// TIA Portal project "Process Control 1" (V13)

(* hardware
DEVICE "S71500/ET200MP station_1"  S7-1500 station
   slot 0: "导轨_0"  6ES7 590-1***0-0AA0
   slot 1: "PLC_1"  CPU 1516-3 PN/DP  6ES7 516-3AN00-0AB0  V1.8
   slot 2: "DI 32x24VDC HF_1"  DI 32x24VDC HF  6ES7 521-1BL00-0AB0  V2.0
   slot 3: "DQ 32x24VDC/0.5A ST_1"  DQ 32x24VDC/0.5A ST  6ES7 522-1BL00-0AB0  V2.0
   slot 4: "AI 8xU/I/RTD/TC ST_1"  AI 8xU/I/RTD/TC ST  6ES7 531-7KF00-0AB0  V2.0
   slot 5: "AQ 4xU/I ST_1"  AQ 4xU/I ST  6ES7 532-5HD00-0AB0  V2.0
DEVICE "PC-System_1"  SIMATIC PC station
   slot 0: "SIMATIC PC station"  Rail  SIMATIC PC-Station  V1.0
      slot 125: "Stationmanager"  Station_Manager  V6.0.4
   slot 1: "HMI_RT_1"  WinCC RT Advanced  6AV2 104-0xxxx-xxxx  13.0.1.0
      slot 33792: "主机接口"  主机接口
   slot 2: "IE general_1"  IE General  IE_CP  V8.2.0
*)

// ===== PLC "PLC_1"  CPU 1516-3 PN/DP =====

VAR_GLOBAL   // PLC tag table "默认变量表"
   "Tag_1" AT %IW4 : Word;
   "Tag_2" AT %MD0 : Real;
   "Tag_3" AT %MD4 : Real;
   "Tag_4" AT %MD8 : Real;
   "Tag_5" AT %MD12 : Real;
   "Tag_6" AT %QW4 : Int;
   "exp_sel01" AT %M16.0 : Bool;
   "exp_sel02" AT %M16.1 : Bool;
   "Tag_7" AT %IW6 : Int;
END_VAR

DATA_BLOCK "TO_WINCC_01"   // DB2
{ S7_Optimized_Access := 'FALSE' }
VERSION : 0.1
   VAR
      Level_Setpoint : Real;
      Level_Feedback : Real;
      Valve_Output : Real;
      Input_sel : Bool;
      ManualValue : Real;
      PID_Reset : Bool;
      PID_Mode : Int;
      Gain : Real;
      Ti : Real;
      Td : Real;
      exp_sel01 : Bool;
      exp_sel02 : Bool;
      Auto_state : Bool;
      Manual_state : Bool;
      Manual_Auto : Bool;
   END_VAR
BEGIN
END_DATA_BLOCK

DATA_BLOCK "TO_WINCC_02"   // DB3
{ S7_Optimized_Access := 'FALSE' }
VERSION : 0.1
   VAR
      Gain_内环 : Real;
      Ti_内环 : Real;
      Gain_外环 : Real;
      Ti_外环 : Real;
      Td_外环 : Real;
   END_VAR
BEGIN
END_DATA_BLOCK

FUNCTION "过控实验1" : Void   // FC1, LAD
{ S7_Optimized_Access := 'FALSE' }
VERSION : 0.1
BEGIN

REGION Network 1: activate peripheral input
   // 选择INPUT或者INPUT_PER参数，为0时是INPUT，为1时是INPUT_PER
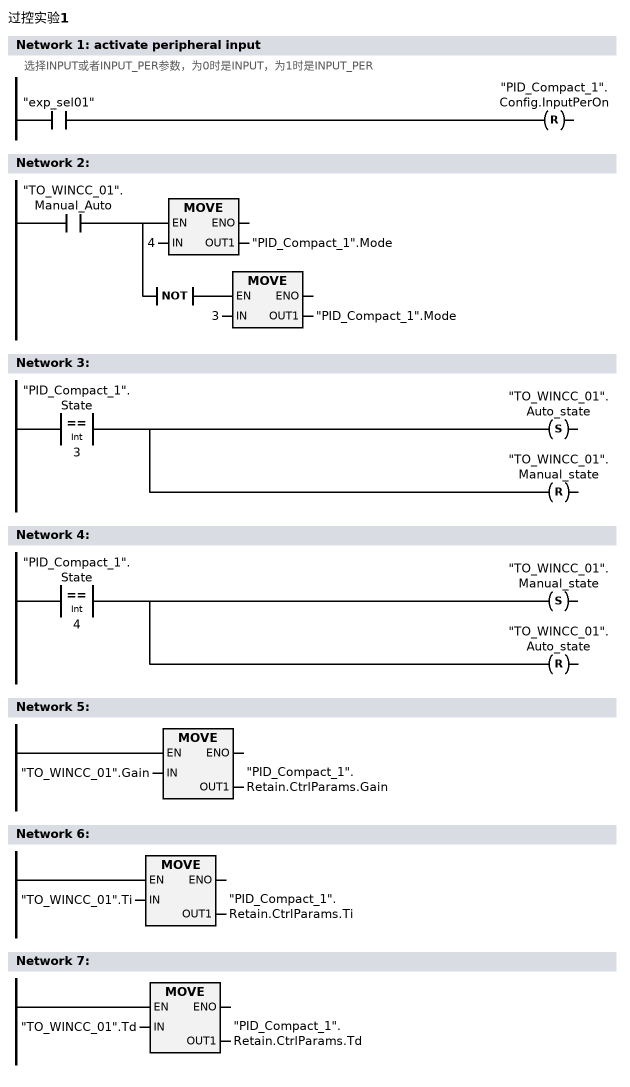
   RUNG wire#powerrail
      Contact( "exp_sel01" )
      R_Coil( "PID_Compact_1".Config.InputPerOn )
   END_RUNG
   // the same network as SCL:
   IF "exp_sel01" THEN "PID_Compact_1".Config.InputPerOn := FALSE; END_IF;
END_REGION

REGION Network 2
   RUNG wire#powerrail
      Contact( "TO_WINCC_01".Manual_Auto )
      wire#w1
      Move(in := 4, out1 => "PID_Compact_1".Mode)
   END_RUNG
   RUNG wire#w1
      Not()
      Move(in := 3, out1 => "PID_Compact_1".Mode)
   END_RUNG
   // the same network as SCL:
   IF "TO_WINCC_01".Manual_Auto THEN "PID_Compact_1".Mode := 4; END_IF;
   IF NOT "TO_WINCC_01".Manual_Auto THEN "PID_Compact_1".Mode := 3; END_IF;
END_REGION

REGION Network 3
   RUNG wire#powerrail
      { S7_Templates := "SrcType := Int" } EQ_Contact(in1 := "PID_Compact_1".State, in2 := 3)
      wire#w1
      S_Coil( "TO_WINCC_01".Auto_state )
   END_RUNG
   RUNG wire#w1
      R_Coil( "TO_WINCC_01".Manual_state )
   END_RUNG
   // the same network as SCL:
   IF "PID_Compact_1".State = 3 THEN
       "TO_WINCC_01".Auto_state := TRUE;
       "TO_WINCC_01".Manual_state := FALSE;
   END_IF;
END_REGION

REGION Network 4
   RUNG wire#powerrail
      { S7_Templates := "SrcType := Int" } EQ_Contact(in1 := "PID_Compact_1".State, in2 := 4)
      wire#w1
      S_Coil( "TO_WINCC_01".Manual_state )
   END_RUNG
   RUNG wire#w1
      R_Coil( "TO_WINCC_01".Auto_state )
   END_RUNG
   // the same network as SCL:
   IF "PID_Compact_1".State = 4 THEN
       "TO_WINCC_01".Manual_state := TRUE;
       "TO_WINCC_01".Auto_state := FALSE;
   END_IF;
END_REGION

REGION Network 5
   RUNG wire#powerrail
      Move(in := "TO_WINCC_01".Gain, out1 => "PID_Compact_1".Retain.CtrlParams.Gain)
   END_RUNG
   // the same network as SCL:
   "PID_Compact_1".Retain.CtrlParams.Gain := "TO_WINCC_01".Gain;
END_REGION

REGION Network 6
   RUNG wire#powerrail
      Move(in := "TO_WINCC_01".Ti, out1 => "PID_Compact_1".Retain.CtrlParams.Ti)
   END_RUNG
   // the same network as SCL:
   "PID_Compact_1".Retain.CtrlParams.Ti := "TO_WINCC_01".Ti;
END_REGION

REGION Network 7
   RUNG wire#powerrail
      Move(in := "TO_WINCC_01".Td, out1 => "PID_Compact_1".Retain.CtrlParams.Td)
   END_RUNG
   // the same network as SCL:
   "PID_Compact_1".Retain.CtrlParams.Td := "TO_WINCC_01".Td;
END_REGION
END_FUNCTION

FUNCTION "过控实验2" : Void   // FC2, LAD
{ S7_Optimized_Access := 'FALSE' }
VERSION : 0.1
BEGIN

REGION Network 1: activate peripheral input
   // 选择INPUT或者INPUT_PER参数，为0时是INPUT，为1时是INPUT_PER
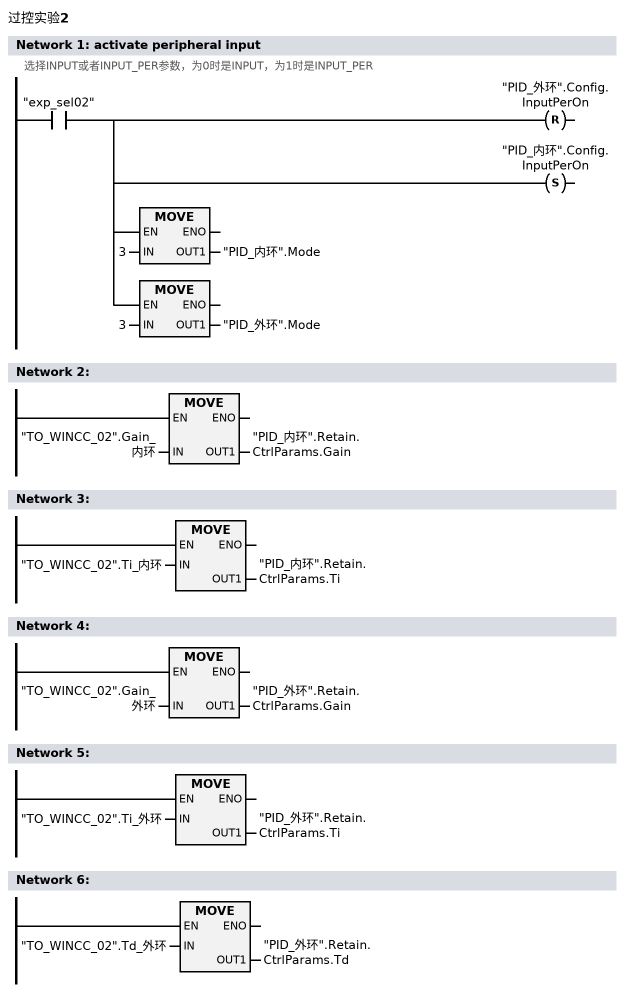
   RUNG wire#powerrail
      Contact( "exp_sel02" )
      wire#w1
      R_Coil( "PID_外环".Config.InputPerOn )
   END_RUNG
   RUNG wire#w1
      S_Coil( "PID_内环".Config.InputPerOn )
   END_RUNG
   RUNG wire#w1
      Move(in := 3, out1 => "PID_内环".Mode)
   END_RUNG
   RUNG wire#w1
      Move(in := 3, out1 => "PID_外环".Mode)
   END_RUNG
   // the same network as SCL:
   IF "exp_sel02" THEN
       "PID_外环".Config.InputPerOn := FALSE;
       "PID_内环".Config.InputPerOn := TRUE;
       "PID_内环".Mode := 3;
       "PID_外环".Mode := 3;
   END_IF;
END_REGION

REGION Network 2
   RUNG wire#powerrail
      Move(in := "TO_WINCC_02".Gain_内环, out1 => "PID_内环".Retain.CtrlParams.Gain)
   END_RUNG
   // the same network as SCL:
   "PID_内环".Retain.CtrlParams.Gain := "TO_WINCC_02".Gain_内环;
END_REGION

REGION Network 3
   RUNG wire#powerrail
      Move(in := "TO_WINCC_02".Ti_内环, out1 => "PID_内环".Retain.CtrlParams.Ti)
   END_RUNG
   // the same network as SCL:
   "PID_内环".Retain.CtrlParams.Ti := "TO_WINCC_02".Ti_内环;
END_REGION

REGION Network 4
   RUNG wire#powerrail
      Move(in := "TO_WINCC_02".Gain_外环, out1 => "PID_外环".Retain.CtrlParams.Gain)
   END_RUNG
   // the same network as SCL:
   "PID_外环".Retain.CtrlParams.Gain := "TO_WINCC_02".Gain_外环;
END_REGION

REGION Network 5
   RUNG wire#powerrail
      Move(in := "TO_WINCC_02".Ti_外环, out1 => "PID_外环".Retain.CtrlParams.Ti)
   END_RUNG
   // the same network as SCL:
   "PID_外环".Retain.CtrlParams.Ti := "TO_WINCC_02".Ti_外环;
END_REGION

REGION Network 6
   RUNG wire#powerrail
      Move(in := "TO_WINCC_02".Td_外环, out1 => "PID_外环".Retain.CtrlParams.Td)
   END_RUNG
   // the same network as SCL:
   "PID_外环".Retain.CtrlParams.Td := "TO_WINCC_02".Td_外环;
END_REGION
END_FUNCTION

FUNCTION "块_1" : Void   // FC3, LAD
{ S7_Optimized_Access := 'FALSE' }
VERSION : 0.1
BEGIN
END_FUNCTION

ORGANIZATION_BLOCK "Main"   // OB1, LAD, ProgramCycle
TITLE = "Main Program Sweep (Cycle)"
{ S7_Optimized_Access := 'FALSE' }
VERSION : 0.1
BEGIN
END_ORGANIZATION_BLOCK

ORGANIZATION_BLOCK "Cyclic interrupt"   // OB30, LAD, CyclicInterrupt
{ S7_Optimized_Access := 'FALSE' }
VERSION : 0.1
   VAR_TEMP   // added for the SCL form of the ladder/FBD networks
      _w1 : Bool;
   END_VAR
BEGIN

REGION Network 1
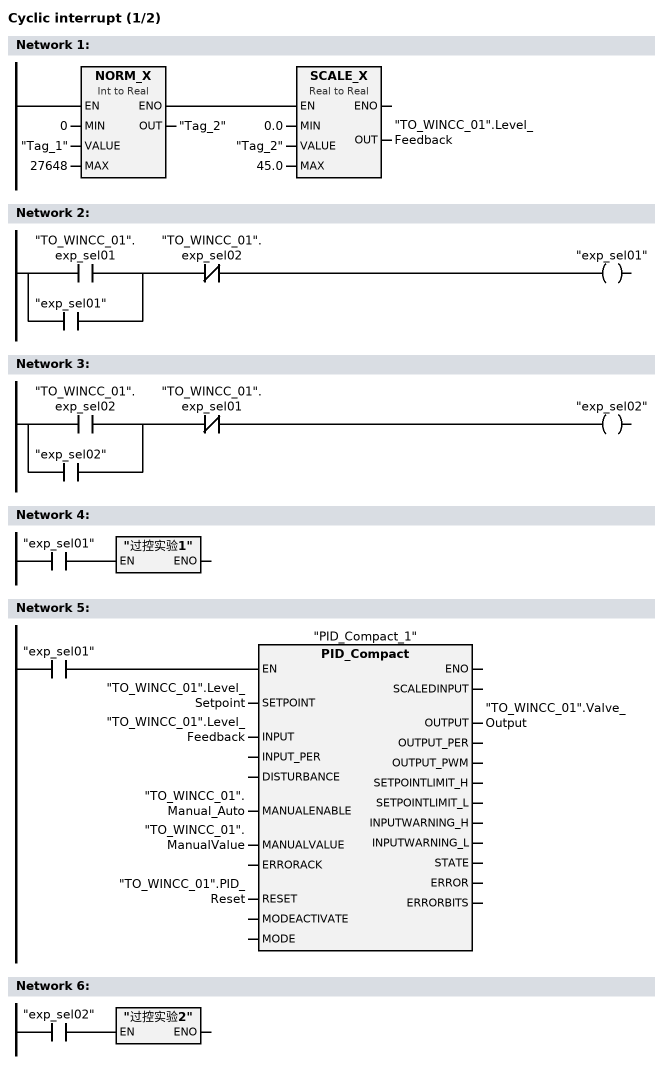
   RUNG wire#powerrail
      { S7_Templates := "[SrcType := Int, DestType := Real]" } Normalize(min := 0, value := "Tag_1", max := 27648, out => "Tag_2")
      { S7_Templates := "[SrcType := Real, DestType := Real]" } Scale(min := 0.0, value := "Tag_2", max := 45.0, out => "TO_WINCC_01".Level_Feedback)
   END_RUNG
   // the same network as SCL:
   "Tag_2" := NORM_X(MIN := 0, VALUE := "Tag_1", MAX := 27648);
   "TO_WINCC_01".Level_Feedback := SCALE_X(MIN := 0.0, VALUE := "Tag_2", MAX := 45.0);
END_REGION

REGION Network 2
   RUNG wire#powerrail
      Contact( "TO_WINCC_01".exp_sel01 )
      wire#w1
      I_Contact( "TO_WINCC_01".exp_sel02 )
      Coil( "exp_sel01" )
   END_RUNG
   RUNG wire#powerrail
      Contact( "exp_sel01" )
   END_RUNG wire#w1
   // the same network as SCL:
   "exp_sel01" := ("TO_WINCC_01".exp_sel01 OR "exp_sel01") AND NOT "TO_WINCC_01".exp_sel02;
END_REGION

REGION Network 3
   RUNG wire#powerrail
      Contact( "TO_WINCC_01".exp_sel02 )
      wire#w1
      I_Contact( "TO_WINCC_01".exp_sel01 )
      Coil( "exp_sel02" )
   END_RUNG
   RUNG wire#powerrail
      Contact( "exp_sel02" )
   END_RUNG wire#w1
   // the same network as SCL:
   "exp_sel02" := ("TO_WINCC_01".exp_sel02 OR "exp_sel02") AND NOT "TO_WINCC_01".exp_sel01;
END_REGION

REGION Network 4
   RUNG wire#powerrail
      Contact( "exp_sel01" )
      "过控实验1"()
   END_RUNG
   // the same network as SCL:
   IF "exp_sel01" THEN "过控实验1"(); END_IF;
END_REGION

REGION Network 5
   IF "exp_sel01" THEN
       "PID_Compact_1"(Setpoint := "TO_WINCC_01".Level_Setpoint,   // PID_Compact
                       Input := "TO_WINCC_01".Level_Feedback,
                       ManualEnable := "TO_WINCC_01".Manual_Auto,
                       ManualValue := "TO_WINCC_01".ManualValue,
                       Reset := "TO_WINCC_01".PID_Reset,
                       Output => "TO_WINCC_01".Valve_Output);
   END_IF;
END_REGION

REGION Network 6
   RUNG wire#powerrail
      Contact( "exp_sel02" )
      "过控实验2"()
   END_RUNG
   // the same network as SCL:
   IF "exp_sel02" THEN "过控实验2"(); END_IF;
END_REGION

REGION Network 7
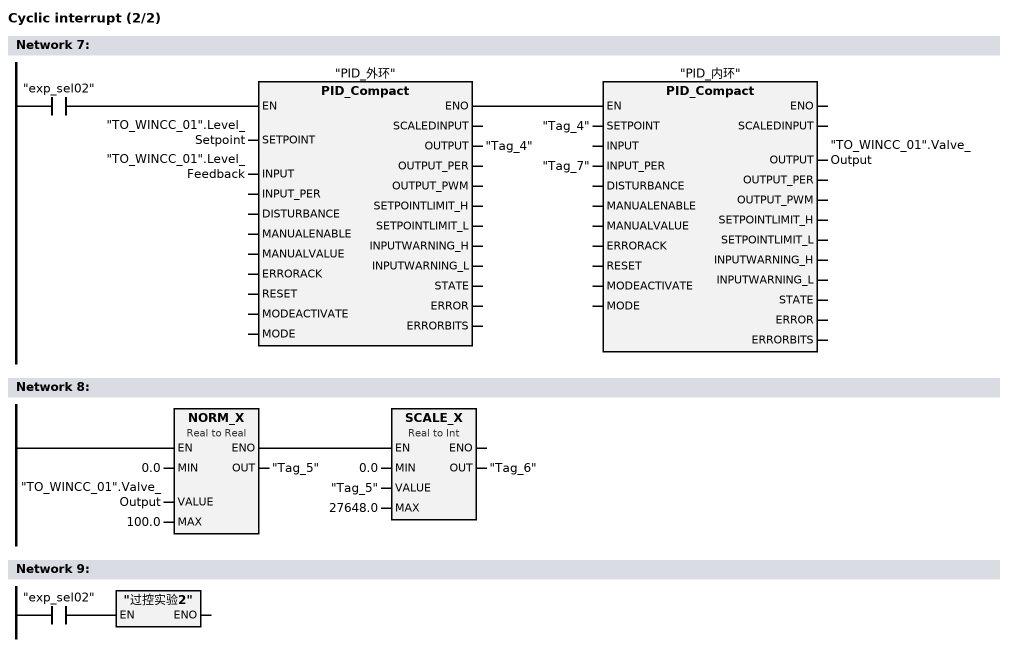
   // ENO of a box is taken as its EN; it also drops when the box reports an error
   #_w1 := "exp_sel02";
   IF #_w1 THEN
       "PID_外环"(Setpoint := "TO_WINCC_01".Level_Setpoint, Input := "TO_WINCC_01".Level_Feedback, Output => "Tag_4");   // PID_Compact
       "PID_内环"(Setpoint := "Tag_4", Input_PER := "Tag_7", Output => "TO_WINCC_01".Valve_Output);   // PID_Compact
   END_IF;
END_REGION

REGION Network 8
   RUNG wire#powerrail
      { S7_Templates := "[SrcType := Real, DestType := Real]" } Normalize(min := 0.0, value := "TO_WINCC_01".Valve_Output, max := 100.0, out => "Tag_5")
      { S7_Templates := "[SrcType := Real, DestType := Int]" } Scale(min := 0.0, value := "Tag_5", max := 27648.0, out => "Tag_6")
   END_RUNG
   // the same network as SCL:
   "Tag_5" := NORM_X(MIN := 0.0, VALUE := "TO_WINCC_01".Valve_Output, MAX := 100.0);
   "Tag_6" := SCALE_X(MIN := 0.0, VALUE := "Tag_5", MAX := 27648.0);
END_REGION

REGION Network 9
   RUNG wire#powerrail
      Contact( "exp_sel02" )
      "过控实验2"()
   END_RUNG
   // the same network as SCL:
   IF "exp_sel02" THEN "过控实验2"(); END_IF;
END_REGION
END_ORGANIZATION_BLOCK

(* ===== HMI "HMI_RT_1" =====
connection "HMI_连接_1": ETHERNET, S7_1500_OMS

HMI tags "默认变量表"
   "TO_WINCC_exp_sel01" : Bool, 100 ms
   "TO_WINCC_exp_sel02" : Bool, 100 ms
   "TO_WINCC_Level_Setpoint" : Real, 100 ms
   "TO_WINCC_Level_Feedback" : Real, 100 ms
   "TO_WINCC_Gain" : Real, 100 ms
   "TO_WINCC_Manual_Auto" : Bool, 100 ms
   "TO_WINCC_ManualValue" : Real, 100 ms
   "TO_WINCC_Manual_state" : Bool, 100 ms
   "TO_WINCC_Auto_state" : Bool, 100 ms
   "TO_WINCC_Ti" : Real, 100 ms
   "TO_WINCC_Td" : Real, 100 ms
   "TO_WINCC_Valve_Output" : Real, 100 ms
   "TO_WINCC_02_Gain_内环" : Real, 100 ms
   "TO_WINCC_02_Ti_内环" : Real, 100 ms
   "TO_WINCC_02_Gain_外环" : Real, 100 ms
   "TO_WINCC_02_Ti_外环" : Real, 100 ms
   "TO_WINCC_02_Td_外环" : Real, 100 ms
   "Tag_4" : Real = PLC "Tag_4", 100 ms
   "Tag_7" : Int = PLC "Tag_7", 100 ms
   "exp_sel01" : Bool = PLC "exp_sel01", 100 ms
   "exp_sel02" : Bool = PLC "exp_sel02", 100 ms

screen "实验选择主画面" 1600x1200
   TextField "文本域_1" at 326,82 size 878x101
   Button "按钮_1" at 498,276 size 562x118
   Button "按钮_2" at 498,501 size 562x118
   TextField "文本域_2" at 390,730 size 785x68

screen "实验1" 1600x1200
   TextField "文本域_1" at 595,12 size 338x40
   TextField "文本域_2" at 27,84 size 150x31
   IOField "I/O 域_1" at 187,80 size 165x36
   TextField "文本域_3" at 414,81 size 150x31
   IOField "I/O 域_2" at 590,79 size 165x36
   TextField "文本域_4" at 126,129 size 49x31
   IOField "I/O 域_3" at 187,126 size 165x36
   TextField "文本域_5" at 1196,30 size 20x31
   Button "按钮_1" at 1268,125 size 230x36
   TextField "文本域_6" at 1249,79 size 137x31
   TextField "文本域_7" at 1389,79 size 63x31
   TextField "文本域_8" at 1196,29 size 150x31
   IOField "I/O 域_4" at 1375,28 size 165x36
   TextField "文本域_9" at 1451,79 size 63x31
   TextField "文本域_10" at 1388,79 size 63x31
   TextField "文本域_11" at 442,129 size 123x31
   IOField "I/O 域_5" at 590,124 size 165x36
   TextField "文本域_12" at 924,128 size 49x31
   IOField "I/O 域_6" at 1002,124 size 165x36
   TrendView "趋势视图_1" at 15,195 size 1562x614
   TextField "文本域_13" at 824,80 size 150x31
   IOField "I/O 域_7" at 1001,78 size 165x36
   TextField "文本域_14" at 27,12 size 179x31
   TextField "文本域_15" at 27,12 size 179x31

screen "实验2" 1600x1200
   TextField "文本域_1" at 595,10 size 338x40
   TextField "文本域_14" at 206,83 size 150x31
   IOField "I/O 域_8" at 366,79 size 165x36
   TextField "文本域_15" at 593,82 size 150x31
   IOField "I/O 域_9" at 769,78 size 165x36
   TextField "文本域_2" at 1004,79 size 150x31
   IOField "I/O 域_1" at 1181,77 size 165x36
   TextField "文本域_3" at 247,137 size 107x31
   IOField "I/O 域_2" at 366,134 size 165x36
   TextField "文本域_4" at 563,137 size 181x31
   IOField "I/O 域_3" at 770,134 size 165x36
   TextField "文本域_5" at 249,191 size 107x31
   IOField "I/O 域_4" at 367,188 size 165x36
   TextField "文本域_6" at 565,191 size 181x31
   IOField "I/O 域_5" at 771,188 size 165x36
   TextField "文本域_7" at 1047,191 size 107x31
   IOField "I/O 域_6" at 1183,187 size 165x36
   TrendView "趋势视图_1" at 21,239 size 1543x557
   TextField "文本域_8" at 27,12 size 179x31
   TextField "文本域_9" at 27,12 size 179x31
*)